(* Schneider Machine Expert - Basic project Test_Traffic, file version 3.0.0.0 *)
(* ProjectInformations: Name=Test_Traffic *)

HARDWARE
  Cpu 0: TM221CE16T
  EthernetConfiguration: NetworkName=M221, IpAllocationMode=ByDhcp, IpAddress=192.168.1.10, SubnetMask=255.255.255.0
  SerialLineConfiguration: Baud=Baud19200, Parity=ParityEven, DataBits=DataBits8, StopBits=StopBits1, PhysicalMedium=PhysicalMediumRs485, TransmissionMode=TransmissionModeModbusRtu, SlaveId=1, Addressing=SlaveAddressing
  MastTask: UsePeriodScanMode=false, PeriodScan=100
  FastTask: Period=255
  CpuBehavior: StartingMode=StartAsPreviousState, AutoSaveRamOnEeprom=true, WatchdogPeriod=250

SYMBOLS  (address, symbol, comment, settings)
  %M0       STATE_RED  "Red State"
  %M1       STATE_YELLOW  "Yellow State"
  %M2       STATE_GREEN  "Green State"
  %I0.0     PB_PED
  %Q0.0     RED
  %Q0.1     YELLOW
  %Q0.2     GREEN

POU Test_Traffic
  (* SectionNumber=1 *)

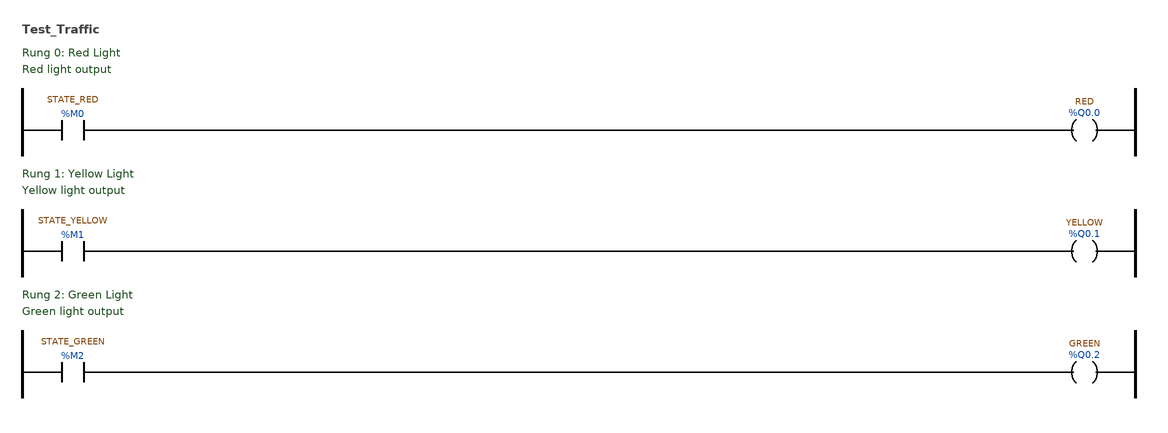

// Rung 0: Red Light
// Red light output
  LD %M0                  (* STATE_RED *)
  ST %Q0.0                (* RED *)
  // as ST:
  //   RED := STATE_RED;

// Rung 1: Yellow Light
// Yellow light output
  LD %M1                  (* STATE_YELLOW *)
  ST %Q0.1                (* YELLOW *)
  // as ST:
  //   YELLOW := STATE_YELLOW;

// Rung 2: Green Light
// Green light output
  LD %M2                  (* STATE_GREEN *)
  ST %Q0.2                (* GREEN *)
  // as ST:
  //   GREEN := STATE_GREEN;
